// LS Electric XG5000 project: 지능형신호(제어)
// PLC LSPLC
// module base 0 slot 0: 입출력 모듈:XBC-DN/DP32H (DC 24V 입력, 트랜지스터 출력 32점 (싱크출력/소스출력))

PROGRAM NewProgram (task: 스캔 프로그램)

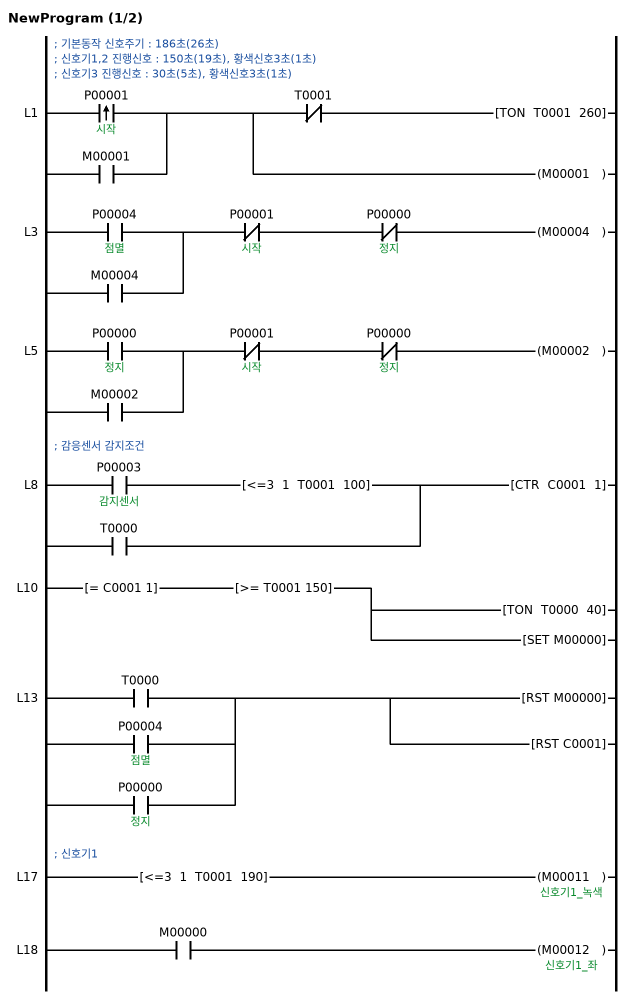
// 기본동작 신호주기 : 186초(26초)
// 신호기1,2 진행신호 : 150초(19초), 황색신호3초(1초)
// 신호기3 진행신호 : 30초(5초), 황색신호3초(1초)
; L1
LOADP     P00001	// 시작
OR        M00001
MPUSH
AND NOT   T0001
TON       T0001 260
MPOP
OUT       M00001
; L3
LOAD      P00004	// 점멸
OR        M00004
AND NOT   P00001	// 시작
AND NOT   P00000	// 정지
OUT       M00004
; L5
LOAD      P00000	// 정지
OR        M00002
AND NOT   P00001	// 시작
AND NOT   P00000	// 정지
OUT       M00002
// 감응센서 감지조건
; L8
LOAD      P00003	// 감지센서
AND<=3    1 T0001 100
OR        T0000
CTR       C0001 1
; L10
LOAD=     C0001 1
AND>=     T0001 150
TON       T0000 40
SET       M00000
; L13
LOAD      T0000
OR        P00004	// 점멸
OR        P00000	// 정지
RST       M00000
RST       C0001
// 신호기1
; L17
LOAD<=3   1 T0001 190
OUT       M00011	// 신호기1_녹색
; L18
LOAD      M00000
OUT       M00012	// 신호기1_좌

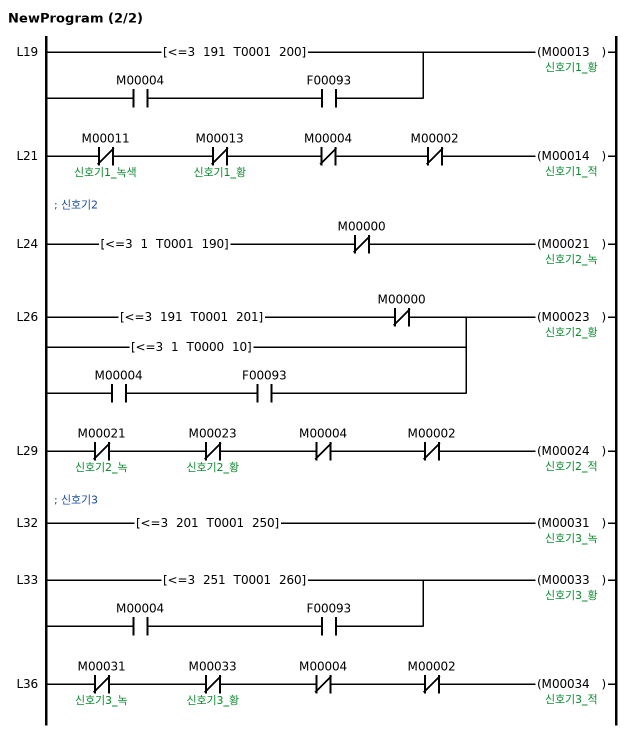
; L19
LOAD<=3   191 T0001 200
LOAD      M00004
AND       F00093
OR LOAD
OUT       M00013	// 신호기1_황
; L21
LOAD NOT  M00011	// 신호기1_녹색
AND NOT   M00013	// 신호기1_황
AND NOT   M00004
AND NOT   M00002
OUT       M00014	// 신호기1_적
// 신호기2
; L24
LOAD<=3   1 T0001 190
AND NOT   M00000
OUT       M00021	// 신호기2_녹
; L26
LOAD<=3   191 T0001 201
AND NOT   M00000
OR<=3     1 T0000 10
LOAD      M00004
AND       F00093
OR LOAD
OUT       M00023	// 신호기2_황
; L29
LOAD NOT  M00021	// 신호기2_녹
AND NOT   M00023	// 신호기2_황
AND NOT   M00004
AND NOT   M00002
OUT       M00024	// 신호기2_적
// 신호기3
; L32
LOAD<=3   201 T0001 250
OUT       M00031	// 신호기3_녹
; L33
LOAD<=3   251 T0001 260
LOAD      M00004
AND       F00093
OR LOAD
OUT       M00033	// 신호기3_황
; L36
LOAD NOT  M00031	// 신호기3_녹
AND NOT   M00033	// 신호기3_황
AND NOT   M00004
AND NOT   M00002
OUT       M00034	// 신호기3_적